FUNCTION_BLOCK EL3433SyncData
VAR_INPUT
	pstEL3433Data	: POINTER TO EL3433Measurement;
	pstEL3433IO		: POINTER TO stEL3433_In;
	pstEL3433OutputIndex	: POINTER TO USINT;
END_VAR

VAR
	pTempReal	: POINTER TO REAL;
	nArrayIndex	: DWORD := TO_DWORD(EL3433Index.listStart);
END_VAR

VAR_STAT
	nCounter1	: EL3433Index := EL3433Index.listStart;
END_VAR

FOR nArrayIndex := TO_DWORD(EL3433Index.listStart) TO TO_DWORD(EL3433Index.listEnd) DO
	IF pstEL3433IO^.dIndex = ConstList.aEL3433Indices[nArrayIndex] THEN
		pTempReal := pstEL3433Data+nArrayIndex*SIZEOF(REAL);
		pTempReal^ := TO_REAL(pstEL3433IO^.dVariant) * ConstList.aEL3433IndicesScale[nArrayIndex];
		EXIT;
	END_IF
END_FOR

pstEL3433OutputIndex^ := ConstList.aEL3433Indices[nCounter1];
IF pstEL3433IO^.dIndex = ConstList.aEL3433Indices[nCounter1] THEN
	nCounter1 := nCounter1 + 1;
	IF nCounter1 > EL3433Index.listEnd THEN
		nCounter1 := EL3433Index.listStart;
	END_IF
END_IF

END_FUNCTION_BLOCK

(* stored: Version 1.1.0.1, ProductVersion 3.1.4022.18
   POU EL3433SyncData: Id {24e958b7-7311-4273-8b0d-0592d477e22b}, SpecialFunc None *)
